Staubli VAL3: create_cube.pgx

public program create_cube(point x_pOrigin, point x_pPointX, point x_pPointY, num x_nDistanceZ)
  local trsf l_trsfCopy
  local point l_pPoint
begin
  //
  // build the cube
  // Origin
  if setFrame(x_pOrigin,x_pPointX,x_pPointY,fCube)==0
    bCreate_cube=true
  endIf
  // Distance x y z
  // X AXES
  l_pPoint.trsf=position(x_pPointX,fCube)
  nDistanceX_cube=l_pPoint.trsf.x
  // Y AXES
  l_pPoint.trsf=position(x_pPointY,fCube)
  nDistanceY_cube=l_pPoint.trsf.y
  // Z distance
  nDistanceZ_cube=x_nDistanceZ
end
